(* Logix 5000 project; controller TCP vendor 1 type 14 code 178 rev 35.12; software revision 35.01 *)

TASK MainTask (continuous, watchdog 500 ms) : MainProgram, TCP_Connection
TASK SafetyTask (periodic, rate 20 ms, priority 10, watchdog 20 ms, safety) : SafetyProgram

MODULES
   Local : vendor 1 type 14 code 178 (Compact 0, rev 35.12)
END_MODULES

TYPE MSG_CreateParameters :
STRUCT
   Type : DINT;   // 1 - TCP ; 2 - UPD
   Addr : MSG_SockAddr;   // Address for the Socket
END_STRUCT
END_TYPE

TYPE MSG_OpenConnectionParameters :
STRUCT
   TimeOut : DINT;   // Timeout in milliseconds
   DestAddr : STRING;   // Hostname or IP adress (ex : 10.88.81.10?port=2813 OR name?port=2813)
END_STRUCT
END_TYPE

TYPE MSG_ReadParameters :
STRUCT
   TimeOut : DINT;   // TimeOut in milliseconds
   BufLen : DINT;   // Number of bytes of data to receive
END_STRUCT
END_TYPE

TYPE MSG_ReadResponse :
STRUCT
   FromAddr : MSG_SockAddr;   // A user-defined structure that can contain the address of the device that sends UDP data. This structure is populated from the end device. For TCP or UDP with OpenConnection, this structure is not used and contains all zeros. The TCP connection conveys all remote address information
   BufLen : DINT;   // Contains the number of bytes of data received
   Buf : SINT[484];   // Contains the data. This number must be large enough to contain the maximum amount of data expected. For a standard connection, the maximum is SINT[484]. For a large connection, the maximum is SINT [3984].
END_STRUCT
END_TYPE

TYPE MSG_SockAddr :
STRUCT
   Family : INT;   // Adress Family Must be 2
   Port : INT;   // Port Number - If random needed use 0
   Addr : DINT;   // IP Address - Each Byte are separated for xxx.xxx.xxx.xxx
END_STRUCT
END_TYPE

TYPE MSG_WriteParameters :
STRUCT
   TimeOut : DINT;   // TimeOut in milliseconds
   ToAddr : MSG_SockAddr;   // Structure that contains the address to which to write UDP data. For TCP or UDP with OpenConnection, this structure is not used and contains all zeros. The TCP connection conveys all required remote address information.
   BufLen : DINT;   // Specify the number of bytes of data to write
   Buf : SINT[472];   // Contains the data. This number must be large enough to contain the maximum amount of data expected. For a standard connection, the maximum is SINT[472]. For a large connection, the maximum is SINT [3972].
END_STRUCT
END_TYPE

VAR_GLOBAL   (* controller tags *)
   Destination_Element_Read_Request : MSG_ReadResponse := (FromAddr.Family := 2, Buf[0] := 78, Buf[1] := 75, Buf[2] := 80, Buf[3] := 49, Buf[9] := 1, Buf[12] := 107, Buf[13] := 99, Buf[14] := 111, Buf[21] := 3, Buf[25] := 1, Buf[29] := 1, Buf[34] := 15, Buf[35] := -125, Buf[36] := -20, Buf[37] := -78, Buf[38] := 50, Buf[39] := 54, Buf[40] := 48, Buf[41] := 51, Buf[42] := 48, Buf[43] := 52, Buf[44] := 48, Buf[45] := 53, Buf[46] := 48, Buf[61] := 3, Buf[63] := -115, Buf[64] := 23, Buf[65] := 112, Buf[66] := 19, Buf[67] := -119, Buf[75] := 48, Buf[76] := 7, Buf[77] := -47, Buf[79] := 60, Buf[80] := 107, Buf[81] := 99, Buf[82] := 111, Buf[89] := 3, Buf[91] := 1, Buf[92] := -20, Buf[93] := -95, Buf[94] := 50, Buf[95] := 54, Buf[96] := 48, Buf[97] := 51, Buf[98] := 48, Buf[99] := 52, Buf[100] := 48, Buf[101] := 51, Buf[102] := 51, Buf[117] := 93, Buf[119] := -115, Buf[120] := 2, Buf[121] := 89, Buf[122] := 19, Buf[123] := -119, Buf[126] := 4, Buf[127] := -52, Buf[130] := 5,
        Buf[131] := 8, Buf[132] := 7, Buf[133] := -41, Buf[135] := 60, Buf[136] := 107, Buf[137] := 99, Buf[138] := 111, Buf[145] := 3, Buf[147] := 2, Buf[148] := 107, Buf[149] := 99, Buf[150] := 111, Buf[157] := 3, Buf[159] := 2, Buf[160] := -20, Buf[161] := -95, Buf[162] := 50, Buf[163] := 54, Buf[164] := 48, Buf[165] := 51, Buf[166] := 48, Buf[167] := 52, Buf[168] := 48, Buf[169] := 51, Buf[170] := 51, Buf[185] := 93, Buf[187] := -115, Buf[188] := 2, Buf[189] := 89, Buf[190] := 19, Buf[191] := -119, Buf[194] := 5, Buf[195] := 59, Buf[198] := 5, Buf[199] := 119, Buf[200] := 7, Buf[201] := -41, Buf[203] := 60, Buf[204] := 107, Buf[205] := 99, Buf[206] := 111, Buf[213] := 3, Buf[215] := 3, Buf[216] := 107, Buf[217] := 99, Buf[218] := 111, Buf[225] := 3, Buf[227] := 3, Buf[229] := 4, Buf[233] := 4, Buf[238] := 15, Buf[239] := -125, Buf[240] := -20, Buf[241] := -95, Buf[242] := 50, Buf[243] := 54, Buf[244] := 48, Buf[245] := 51, Buf[246] := 48, Buf[247] := 52,
        Buf[248] := 48, Buf[249] := 51, Buf[250] := 51, Buf[265] := 93, Buf[267] := -115, Buf[268] := 2, Buf[269] := 89, Buf[270] := 19, Buf[271] := -119, Buf[274] := 9, Buf[275] := -13, Buf[278] := 10, Buf[279] := 47, Buf[280] := 7, Buf[281] := -41, Buf[283] := 60, Buf[284] := 107, Buf[285] := 99, Buf[286] := 111, Buf[293] := 3, Buf[295] := 4, Buf[297] := 5, Buf[301] := 5, Buf[306] := 15, Buf[307] := -125, Buf[308] := -20, Buf[309] := -95, Buf[310] := 50, Buf[311] := 54, Buf[312] := 48, Buf[313] := 51, Buf[314] := 48, Buf[315] := 52, Buf[316] := 48, Buf[317] := 51, Buf[318] := 51, Buf[333] := 93, Buf[335] := -115, Buf[336] := 2, Buf[337] := 89, Buf[338] := 19, Buf[339] := -119, Buf[342] := 13, Buf[343] := -50, Buf[346] := 14, Buf[347] := 10, Buf[348] := 7, Buf[349] := -41, Buf[351] := 60, Buf[352] := 107, Buf[353] := 99, Buf[354] := 111, Buf[361] := 3, Buf[363] := 5, Buf[365] := 6, Buf[369] := 6, Buf[374] := 15, Buf[375] := -125, Buf[376] := -20, Buf[377] := -95,
        Buf[378] := 50, Buf[379] := 54, Buf[380] := 48, Buf[381] := 51, Buf[382] := 48, Buf[383] := 52, Buf[384] := 48, Buf[385] := 51, Buf[386] := 51, Buf[401] := 93, Buf[403] := -115, Buf[404] := 2, Buf[405] := 89, Buf[406] := 19, Buf[407] := -119, Buf[410] := 14, Buf[411] := 25, Buf[414] := 14, Buf[415] := 85, Buf[416] := 7, Buf[417] := -41, Buf[419] := 60, Buf[420] := 107, Buf[421] := 99, Buf[422] := 111, Buf[429] := 3, Buf[431] := 6, Buf[433] := 7, Buf[437] := 7, Buf[442] := 15, Buf[443] := -125, Buf[444] := -20, Buf[445] := -95, Buf[446] := 50, Buf[447] := 54, Buf[448] := 48, Buf[449] := 51, Buf[450] := 48, Buf[451] := 52, Buf[452] := 48, Buf[453] := 51, Buf[454] := 51, Buf[469] := 93, Buf[471] := -115, Buf[472] := 2, Buf[473] := 89, Buf[474] := 19, Buf[475] := -119, Buf[478] := 15, Buf[479] := -31, Buf[482] := 16, Buf[483] := 29);
   Destination_Element_Write_Request : DINT := 48;   // Lenght of the Data written
   Destination_Element_Write_Request_Payloa : DINT := 48;   // Lenght of the Data written
   Instance_OPTP : DINT := 21276;
   MSG_Create_Socket : MESSAGE;
        MessageParameters(ServiceCode := 16#004b, LocalElement := Source_Element_Create_Socket, DestinationTag := Instance_OPTP, ...)
   MSG_Delete_All_Socket : MESSAGE;
        MessageParameters(ServiceCode := 16#0051, ...)
   MSG_Open_Connection : MESSAGE;
        MessageParameters(ServiceCode := 16#004c, LocalElement := Source_Element_Open_Connection, ...)
   MSG_Read_Request : MESSAGE;
        MessageParameters(ServiceCode := 16#004d, LocalElement := Source_Element_Read_Request, DestinationTag := Destination_Element_Read_Request, ...)
   MSG_Write_Request : MESSAGE;
        MessageParameters(ServiceCode := 16#004e, LocalElement := Source_Element_Write_Request, DestinationTag := Destination_Element_Write_Request, ...)
   MSG_Write_Request_Payload : MESSAGE;
        MessageParameters(ServiceCode := 16#004e, LocalElement := Source_Element_Write_Request_Payload, DestinationTag := Destination_Element_Write_Request_Payloa, ...)
   Source_Element_Create_Socket : MSG_CreateParameters := (Type := 1, Addr.Family := 2);   // Source parameters for MSG Create Socket
   Source_Element_Open_Connection : MSG_OpenConnectionParameters := (TimeOut := 5000, DestAddr := '192.120.0.203?port=5010$00');
   Source_Element_Read_Request : MSG_ReadParameters := (TimeOut := 3000, BufLen := 484);
   Source_Element_Write_Request : MSG_WriteParameters := (TimeOut := 5000, BufLen := 8, Buf[0] := 78, Buf[1] := 75, Buf[2] := 80, Buf[3] := 49, Buf[4] := 57, Buf[5] := 57, Buf[6] := 57, Buf[7] := 57);
   Source_Element_Write_Request_Payload : MSG_WriteParameters := (TimeOut := 5000, BufLen := 7, Buf[0] := 98, Buf[1] := 105, Buf[2] := 103, Buf[3] := 78, Buf[4] := 75, Buf[5] := 80, Buf[6] := 50);
END_VAR

PROGRAM MainProgram   (* main routine MainRoutine *)

ROUTINE MainRoutine   (* ladder *)
END_ROUTINE
END_PROGRAM

PROGRAM SafetyProgram   (* main routine MainRoutine, safety *)

ROUTINE MainRoutine   (* ladder *)
END_ROUTINE
END_PROGRAM

PROGRAM TCP_Connection   (* main routine Main *)
VAR
   Action_000 : SFC_ACTION := (Status := 16#0020_0000, PauseTimer := 1);
   Action_001 : SFC_ACTION := (Status := 16#0020_0000, PauseTimer := 1);
   Action_002 : SFC_ACTION := (Status := 16#0020_0000, PauseTimer := 1);
   Action_003 : SFC_ACTION := (Status := 16#0020_0000, PauseTimer := 1);
   Action_004 : SFC_ACTION := (Status := 16#0020_0000, PauseTimer := 1);
   Action_005 : SFC_ACTION := (Status := 16#0020_0000, PauseTimer := 1);
   Action_006 : SFC_ACTION := (Status := 16#0020_0000, PauseTimer := 1);
   Action_007 : SFC_ACTION := (Status := 16#0020_0000, PauseTimer := 1);
   Action_008 : SFC_ACTION := (Status := 16#0020_0000, PauseTimer := 1);
   Convert_ok : BOOL;
   FALSE : BOOL; {constant}
   Footer_Invalid : BOOL;
   Footer_Valid : BOOL;   // M
   Header_At_Zero : BOOL;   // M
   Header_Found : BOOL;   // M
   Header_Pos : DINT;   // M B
   Header_Ready : BOOL;   // M
   Header_Send : BOOL;   // M
   Header_Valid : BOOL;   // M
   I_Size_Payload : DINT;   // M B
   ind : DINT;
   Init_Done : BOOL;   // M
   Invalide_Size_Format : BOOL;   // M
   NEKO : BOOL;   // B
   No_Header : BOOL;
   ONS : BOOL[32];
        [0]   // used
        [1]   // used
        [2]   // used
   Open_Connection : BOOL;   // M
   Open_started : BOOL := 1;   // M
   Payload_buffer : SINT[4096];   // M B
   Read_Done : BOOL;   // M
   Request_to_send : BOOL;   // M B
   Reset_Error : BOOL;   // M B
   Rx_Buffer : SINT[4096];   // M B
   Rx_Count : DINT;   // M B
   Rx_Update : BOOL;
   S00_Init : SFC_STEP := (Status := 16#0020_0000, PauseTimer := 1);
   S100_CHECK_FOOTER : SFC_STEP := (Status := 16#0020_0000, PauseTimer := 1);
   S10_IDLE : SFC_STEP := (Status := 16#0020_0000, PauseTimer := 1);
   S110_EXTRACT : SFC_STEP := (Status := 16#0020_0000, PauseTimer := 1);
   S120_PROCESS : SFC_STEP := (Status := 16#0020_0000, PauseTimer := 1);
   S130_RESYNC : SFC_STEP := (Status := 16#0020_0000, PauseTimer := 1);
   S20_Write : SFC_STEP := (Status := 16#0020_0000, PauseTimer := 1);
   S30_WAIT_DATA : SFC_STEP := (Status := 16#0020_0000, PauseTimer := 1);
   S40_APPEND_DATA : SFC_STEP := (Status := 16#0020_0000, PauseTimer := 1);
   S50_FIIND_HEADER : SFC_STEP := (Status := 16#0020_0000, PauseTimer := 1);
   S60_CLEAN_BUFFER : SFC_STEP := (Status := 16#0020_0000, PauseTimer := 1);
   S70_WAIT_HEADER : SFC_STEP := (Status := 16#0020_0000, PauseTimer := 1);
   S80_CHECK_HEADER : SFC_STEP := (Status := 16#0020_0000, PauseTimer := 1);
   S900_ERROR : SFC_STEP := (Status := 16#0020_0000, PauseTimer := 1);
   S90_WAIT_FRAME : SFC_STEP := (Status := 16#0020_0000, PauseTimer := 1);
   Signature_False : BOOL;   // M
   Size_Overflow : BOOL;   // M
   Size_Payload : STRING;   // M B
   Socket_Create : BOOL;   // M
   T00A10 : BOOL;
   T00A900 : BOOL;
   T100A110 : BOOL;
   T100A130 : BOOL;
   T10A20 : BOOL;
   T110A120 : BOOL;
   T120A10 : BOOL;
   T120A50 : BOOL;
   T130A30 : BOOL;
   T130A50 : BOOL;
   T20A30 : BOOL;
   T20A900 : BOOL;
   T30A40 : BOOL;
   T30A401 : BOOL;
   T30A900 : BOOL;
   T40A50 : BOOL;
   T50A30 : BOOL;
   T50A60 : BOOL;
   T50A70 : BOOL;
   T60A80 : BOOL;
   T70A30 : BOOL;
   T70A80 : BOOL;
   T80A130 : BOOL;
   T80A90 : BOOL;
   T900A00 : BOOL;
   T90A100 : BOOL;
   T90A30 : BOOL;
   TRUE : BOOL := 1; {constant}
   Write_Done : BOOL;   // M
END_VAR

ROUTINE Graphe_Etat   (* sequential function chart *)
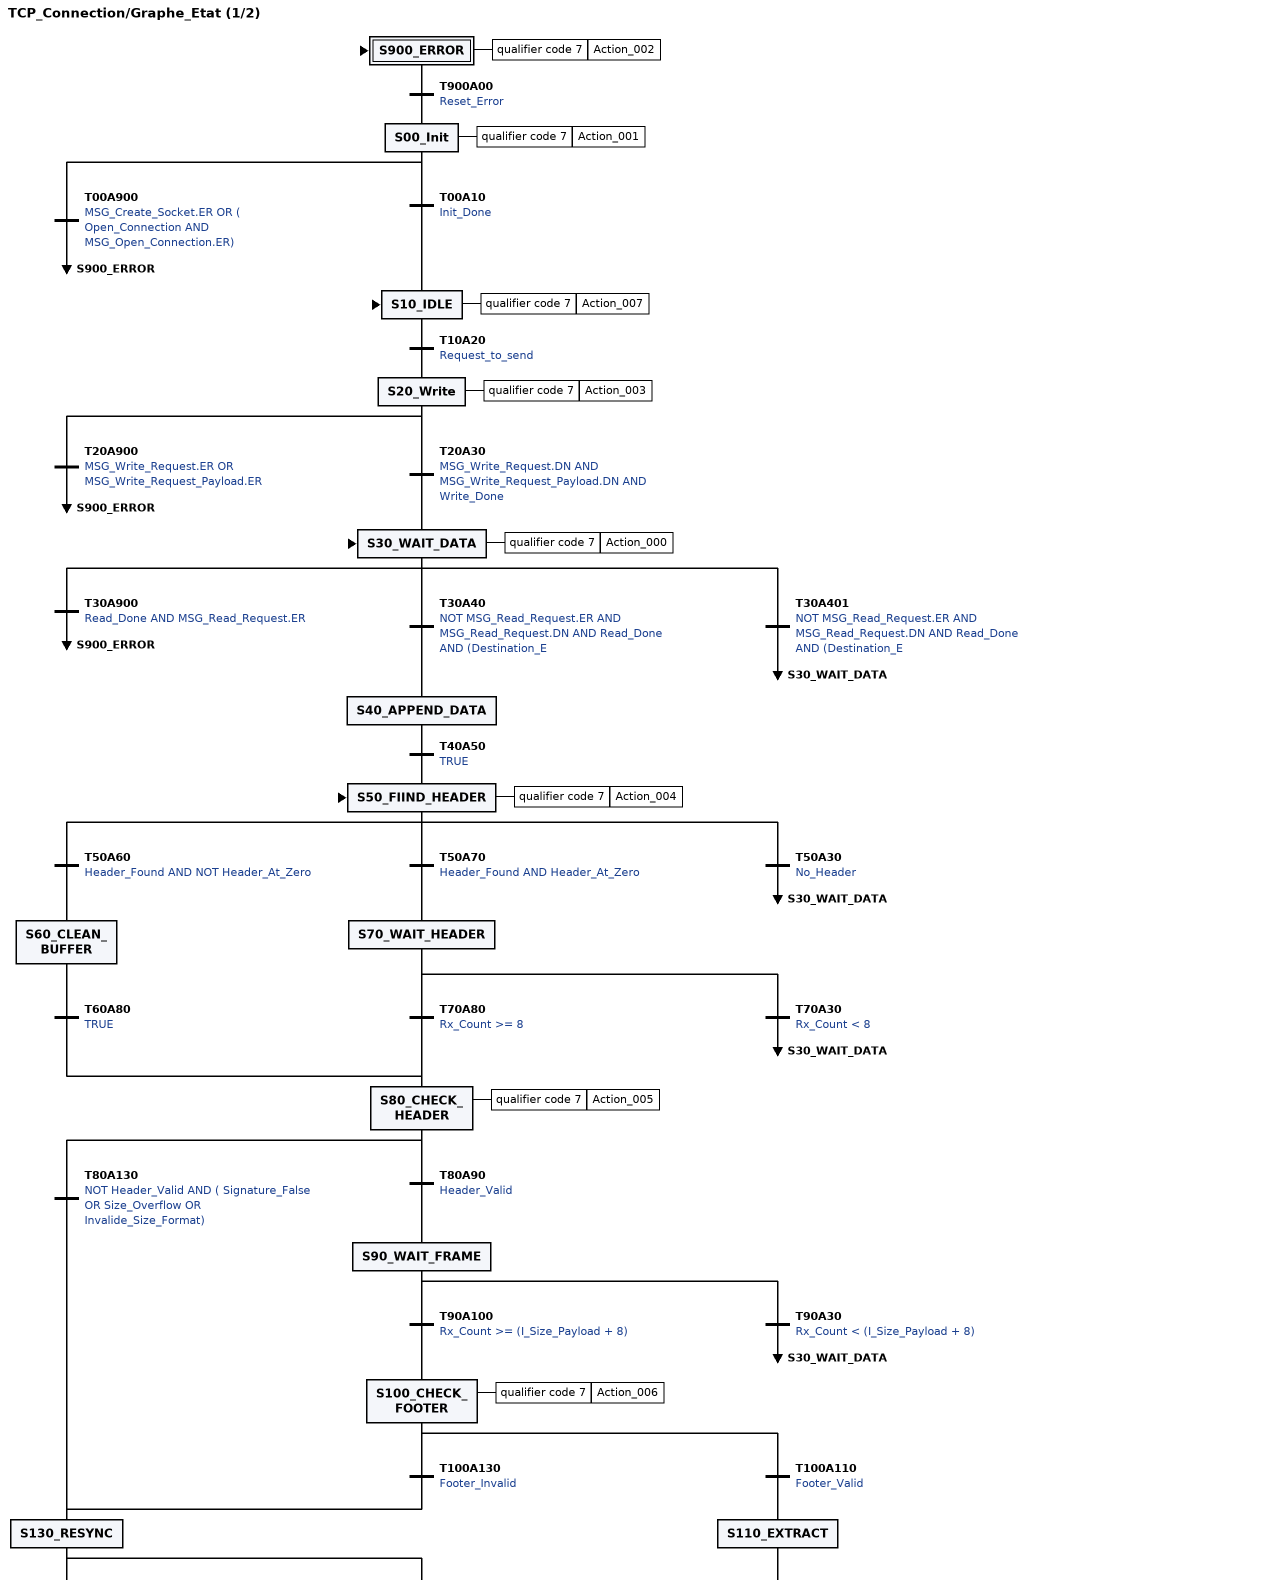
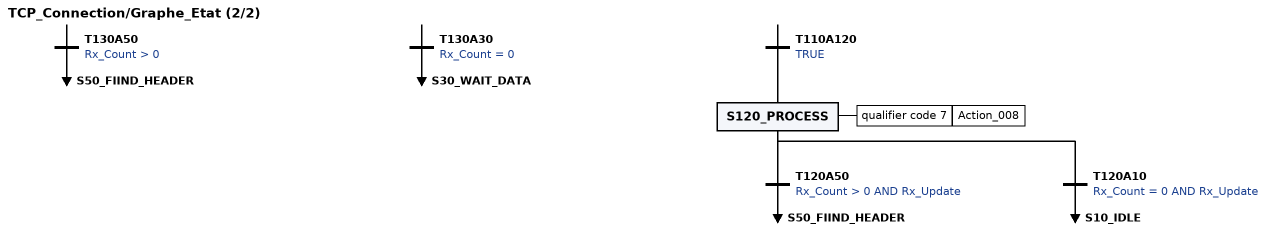
   // RESET ALL
   INITIAL_STEP S900_ERROR:
      ACTION Action_002 (qualifier code 7):
         Reset_Error := 0;
      END_ACTION
   END_STEP
   TRANSITION T900A00 FROM S900_ERROR TO S00_Init
      := Reset_Error
   END_TRANSITION
   STEP S00_Init:
      ACTION Action_001 (qualifier code 7):
         Socket_Create := 0;
         Open_started := 0;
         Open_Connection := 0;
         Init_Done := 0;
      END_ACTION
   END_STEP
   TRANSITION T00A900 FROM S00_Init TO S900_ERROR
      := MSG_Create_Socket.ER OR (
         Open_Connection AND
         MSG_Open_Connection.ER)
   END_TRANSITION
   TRANSITION T00A10 FROM S00_Init TO S10_IDLE
      := Init_Done
   END_TRANSITION
   STEP S10_IDLE:
      ACTION Action_007 (qualifier code 7):
         Rx_Count := 0;
         Request_to_send := 0;
      END_ACTION
   END_STEP
   TRANSITION T10A20 FROM S10_IDLE TO S20_Write
      := Request_to_send
   END_TRANSITION
   STEP S20_Write:
      ACTION Action_003 (qualifier code 7):
         Convert_ok := 0;
         Header_Send := 0;
         Write_Done := 0;
      END_ACTION
   END_STEP
   TRANSITION T20A900 FROM S20_Write TO S900_ERROR
      := MSG_Write_Request.ER OR
         MSG_Write_Request_Payload.ER
   END_TRANSITION
   TRANSITION T20A30 FROM S20_Write TO S30_WAIT_DATA
      := MSG_Write_Request.DN AND
         MSG_Write_Request_Payload.DN AND
         Write_Done
         
   END_TRANSITION
   STEP S30_WAIT_DATA:
      ACTION Action_000 (qualifier code 7):
         Read_Done := 0;
         Destination_Element_Read_Request.BufLen :=0;
      END_ACTION
   END_STEP
   TRANSITION T30A40 FROM S30_WAIT_DATA TO S40_APPEND_DATA
      := NOT MSG_Read_Request.ER AND
         MSG_Read_Request.DN AND
         Read_Done AND
         (Destination_Element_Read_Request.BufLen > 0)
   END_TRANSITION
   TRANSITION T30A401 FROM S30_WAIT_DATA TO S30_WAIT_DATA
      := NOT MSG_Read_Request.ER AND
         MSG_Read_Request.DN AND
         Read_Done AND
         (Destination_Element_Read_Request.BufLen = 0)
   END_TRANSITION
   TRANSITION T30A900 FROM S30_WAIT_DATA TO S900_ERROR
      := Read_Done AND
         MSG_Read_Request.ER
   END_TRANSITION
   STEP S40_APPEND_DATA:
   END_STEP
   TRANSITION T40A50 FROM S40_APPEND_DATA TO S50_FIIND_HEADER
      := TRUE
         
   END_TRANSITION
   STEP S50_FIIND_HEADER:
      ACTION Action_004 (qualifier code 7):
         Header_Found := 0;
         Header_At_Zero := 0;
         Header_Pos := 0;
         No_Header := 0;
      END_ACTION
   END_STEP
   TRANSITION T50A60 FROM S50_FIIND_HEADER TO S60_CLEAN_BUFFER
      := Header_Found AND NOT
         Header_At_Zero
   END_TRANSITION
   TRANSITION T50A70 FROM S50_FIIND_HEADER TO S70_WAIT_HEADER
      := Header_Found AND
         Header_At_Zero
         
         
   END_TRANSITION
   TRANSITION T50A30 FROM S50_FIIND_HEADER TO S30_WAIT_DATA
      := No_Header
   END_TRANSITION
   STEP S60_CLEAN_BUFFER:
   END_STEP
   STEP S70_WAIT_HEADER:
   END_STEP
   TRANSITION T60A80 FROM S60_CLEAN_BUFFER TO S80_CHECK_HEADER
      := TRUE
   END_TRANSITION
   TRANSITION T70A80 FROM S70_WAIT_HEADER TO S80_CHECK_HEADER
      := Rx_Count >= 8
   END_TRANSITION
   TRANSITION T70A30 FROM S70_WAIT_HEADER TO S30_WAIT_DATA
      := Rx_Count < 8
   END_TRANSITION
   STEP S80_CHECK_HEADER:
      ACTION Action_005 (qualifier code 7):
         Invalide_Size_Format := 0;
         Size_Overflow := 0;
         Header_Valid := 0;
         Signature_False := 0;
      END_ACTION
   END_STEP
   TRANSITION T80A130 FROM S80_CHECK_HEADER TO S130_RESYNC
      := NOT Header_Valid AND (
         Signature_False OR
         Size_Overflow OR
         Invalide_Size_Format)
   END_TRANSITION
   TRANSITION T80A90 FROM S80_CHECK_HEADER TO S90_WAIT_FRAME
      := Header_Valid
   END_TRANSITION
   STEP S90_WAIT_FRAME:
   END_STEP
   TRANSITION T90A30 FROM S90_WAIT_FRAME TO S30_WAIT_DATA
      := Rx_Count < (I_Size_Payload + 8)
   END_TRANSITION
   TRANSITION T90A100 FROM S90_WAIT_FRAME TO S100_CHECK_FOOTER
      := Rx_Count >= (I_Size_Payload + 8)
   END_TRANSITION
   STEP S100_CHECK_FOOTER:
      ACTION Action_006 (qualifier code 7):
         Footer_Valid := 0;
         Footer_Invalid := 0;
      END_ACTION
   END_STEP
   TRANSITION T100A130 FROM S100_CHECK_FOOTER TO S130_RESYNC
      := Footer_Invalid
   END_TRANSITION
   TRANSITION T100A110 FROM S100_CHECK_FOOTER TO S110_EXTRACT
      := Footer_Valid
   END_TRANSITION
   STEP S130_RESYNC:
   END_STEP
   STEP S110_EXTRACT:
   END_STEP
   TRANSITION T130A50 FROM S130_RESYNC TO S50_FIIND_HEADER
      := Rx_Count > 0
   END_TRANSITION
   TRANSITION T130A30 FROM S130_RESYNC TO S30_WAIT_DATA
      := Rx_Count = 0
   END_TRANSITION
   TRANSITION T110A120 FROM S110_EXTRACT TO S120_PROCESS
      := TRUE
   END_TRANSITION
   STEP S120_PROCESS:
      ACTION Action_008 (qualifier code 7):
         Rx_Update := 0;
      END_ACTION
   END_STEP
   TRANSITION T120A50 FROM S120_PROCESS TO S50_FIIND_HEADER
      := Rx_Count > 0 AND
         Rx_Update
   END_TRANSITION
   TRANSITION T120A10 FROM S120_PROCESS TO S10_IDLE
      := Rx_Count = 0 AND
         Rx_Update
         
   END_TRANSITION
END_ROUTINE

ROUTINE Main   (* ladder *)
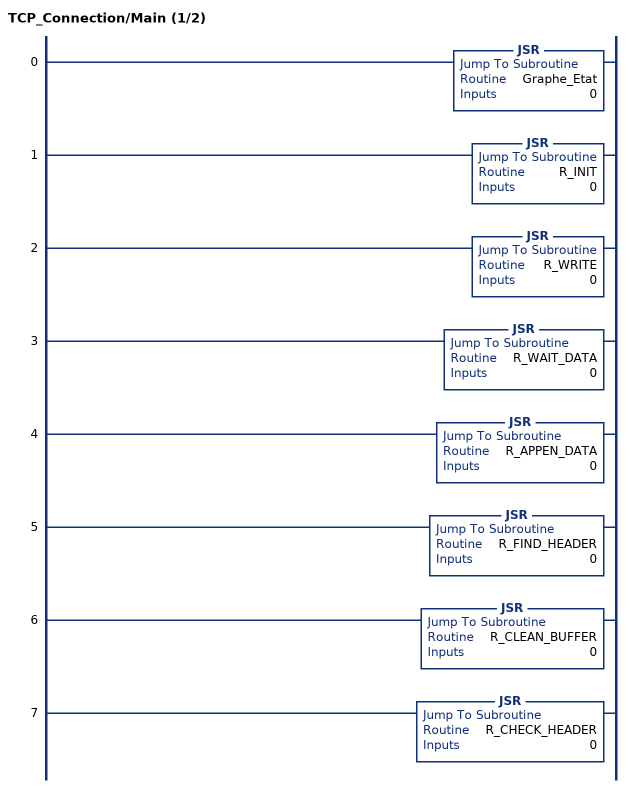
   0: JSR(Graphe_Etat,0);
   1: JSR(R_INIT,0);
   2: JSR(R_WRITE,0);
   3: JSR(R_WAIT_DATA,0);
   4: JSR(R_APPEN_DATA,0);
   5: JSR(R_FIND_HEADER,0);
   6: JSR(R_CLEAN_BUFFER,0);
   7: JSR(R_CHECK_HEADER,0);
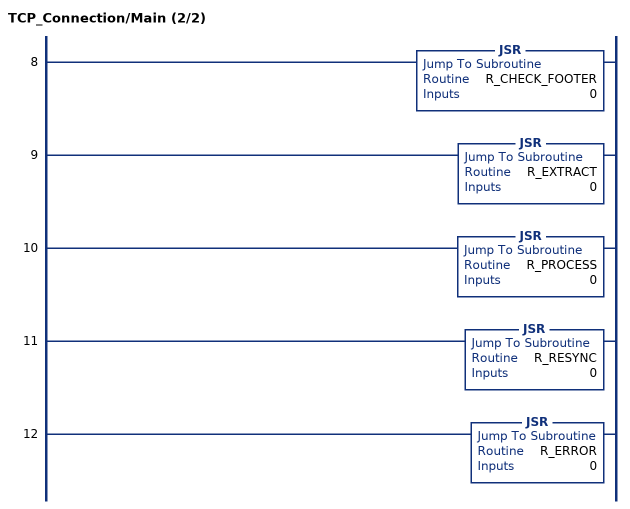
   8: JSR(R_CHECK_FOOTER,0);
   9: JSR(R_EXTRACT,0);
   10: JSR(R_PROCESS,0);
   11: JSR(R_RESYNC,0);
   12: JSR(R_ERROR,0);
END_ROUTINE

ROUTINE R_APPEN_DATA   (* structured text *)
   IF S40_APPEND_DATA.SA THEN
   	for ind := 0 to (Destination_Element_Read_Request.BufLen - 1) do
   		Rx_Buffer[Rx_Count + ind] := Destination_Element_Read_Request.Buf[ind];
   	end_for;
   	Rx_Count := Rx_Count + Destination_Element_Read_Request.BufLen;
   ELSE
   END_IF;
END_ROUTINE

ROUTINE R_CHECK_FOOTER   (* structured text *)
   IF S100_CHECK_FOOTER.SA THEN
   	IF Rx_Buffer[Rx_Count - 4] = 78 AND Rx_Buffer[Rx_Count - 3] = 75 AND
   	   Rx_Buffer[Rx_Count - 2] = 80 AND Rx_Buffer[Rx_Count - 1] = 50 THEN
   	   Footer_Valid := 1;
   	   Footer_Invalid := 0;
   
   	ELSE
   		Footer_Invalid := 1;
   		Footer_Valid := 0;
   	END_IF;
   ELSE
   
   END_IF;
   
END_ROUTINE

ROUTINE R_CHECK_HEADER   (* structured text *)
   IF S80_CHECK_HEADER.SA THEN
   	IF Rx_Buffer[0] = 78 AND Rx_Buffer[1] = 75 AND Rx_Buffer[2] = 80 AND Rx_Buffer[3] = 49 THEN
   		FOR ind := 4 TO 7 DO
   			Size_Payload.DATA[ind - 4] := Rx_Buffer[ind];
   		END_FOR;
   		Size_Payload.LEN := 4;
   
   		// Copy into a STRING buffer for convertion purpuse
   		FOR ind := 0 TO 3 DO
   			//Check that the ASCII format refer to a number
   			IF Size_Payload.DATA[ind] > 57 OR Size_Payload.DATA[ind] < 48 THEN
   				Invalide_Size_Format := 1;
   				EXIT;
   			ELSE
   				Invalide_Size_Format := 0;
   			END_IF;
   		END_FOR;
   		IF NOT Invalide_Size_Format THEN
   			//Convert to a DINT then we check that the size is not bigger than our Rx_Buffer
   			STOD(Size_Payload, I_Size_Payload);
   			IF I_Size_Payload > 4096 THEN
   				Size_Overflow := 1;
   				Header_Valid := 0;
   			ELSE
   				Size_Overflow := 0;
   				Header_Valid := 1;
   			END_IF;
   		ELSE
   			// Nothing to do because invalide format
   		END_IF;
   	ELSE
   		Signature_False := 1;
   	END_IF;
   ELSE
   
   END_IF;
END_ROUTINE

ROUTINE R_CLEAN_BUFFER   (* structured text *)
   IF S60_CLEAN_BUFFER.FS THEN
   	FOR ind := 0 TO (Rx_Count - 1 - Header_Pos) DO
   		Rx_Buffer[ind] := Rx_Buffer[Header_Pos + ind];
   	END_FOR;
   	Rx_Count := Rx_Count - Header_Pos;
   ELSE
   
   END_IF;
END_ROUTINE

ROUTINE R_ERROR   (* ladder *)
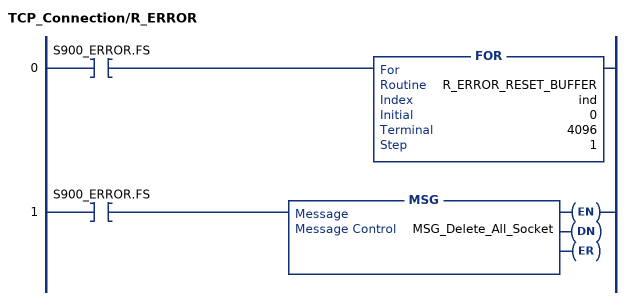
   0: XIC(S900_ERROR.FS)FOR(R_ERROR_RESET_BUFFER,ind,0,4096,1);
   1: XIC(S900_ERROR.FS)MSG(MSG_Delete_All_Socket);
END_ROUTINE

ROUTINE R_ERROR_RESET_BUFFER   (* ladder *)
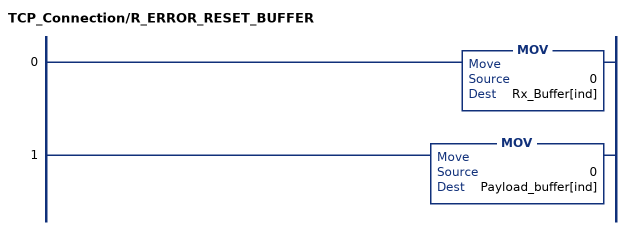
   0: MOV(0,Rx_Buffer[ind]);
   1: MOV(0,Payload_buffer[ind]);
END_ROUTINE

ROUTINE R_EXTRACT   (* structured text *)
   IF S110_EXTRACT.SA THEN
   	FOR ind := 0 TO (Rx_Count - 8 - 4 - 1) DO  //8 for header 4 for footer
   		Payload_buffer[ind] := Rx_Buffer[8 + ind];
   	END_FOR;
   ELSE
   
   END_IF;
END_ROUTINE

ROUTINE R_FIND_HEADER   (* structured text *)
   IF S50_FIIND_HEADER.SA THEN
   	FOR ind := 0 TO (Rx_Count - 4) DO
   		IF Rx_Buffer[ind] = 78 AND Rx_Buffer[ind + 1] = 75 AND Rx_Buffer[ind + 2] = 80 AND Rx_Buffer[ind + 3] = 49 THEN
   			Header_Found := 1;
   			No_Header := 0;
   			Header_Pos := ind;
   			IF Header_Pos = 0 THEN
   				Header_At_Zero := 1;
   			END_IF;
   			EXIT;
   		ELSE
   
   		END_IF;
   	END_FOR;
   	IF ind >= (Rx_Count - 4) then
   		Header_Found := 0;
   		No_Header := 1;
   	END_IF;
   ELSE
   
   END_IF;
END_ROUTINE

ROUTINE R_INIT   (* ladder *)
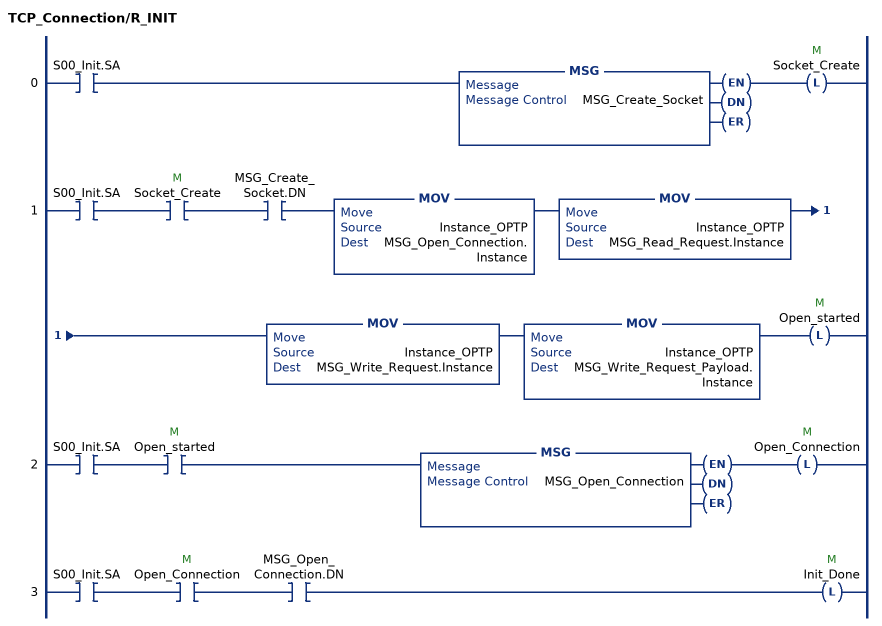
   0: XIC(S00_Init.SA)MSG(MSG_Create_Socket)OTL(Socket_Create);
   1: XIC(S00_Init.SA)XIC(Socket_Create)XIC(MSG_Create_Socket.DN)MOV(Instance_OPTP,MSG_Open_Connection.Instance)MOV(Instance_OPTP,MSG_Read_Request.Instance)MOV(Instance_OPTP,MSG_Write_Request.Instance)MOV(Instance_OPTP,MSG_Write_Request_Payload.Instance)OTL(Open_started);
   2: XIC(S00_Init.SA)XIC(Open_started)MSG(MSG_Open_Connection)OTL(Open_Connection);
   3: XIC(S00_Init.SA)XIC(Open_Connection)XIC(MSG_Open_Connection.DN)OTL(Init_Done);
END_ROUTINE

ROUTINE R_PROCESS   (* structured text *)
   //No DATA to process now
   IF S120_PROCESS.SA AND NOT Rx_Update THEN
   	Rx_Count := Rx_Count - 8 - I_Size_Payload;
   	Rx_Update := 1;
   ELSE
   END_iF;
END_ROUTINE

ROUTINE R_RESYNC   (* structured text *)
   IF S130_RESYNC.FS THEN
   
   ELSE
   
   END_IF;
END_ROUTINE

ROUTINE R_WAIT_DATA   (* ladder *)
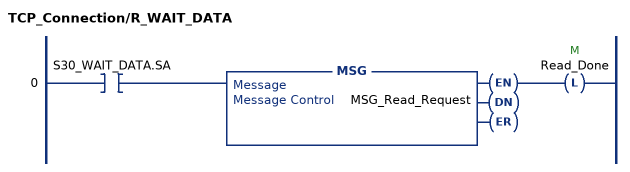
   0: XIC(S30_WAIT_DATA.SA)MSG(MSG_Read_Request)OTL(Read_Done);
END_ROUTINE

ROUTINE R_WRITE   (* ladder *)
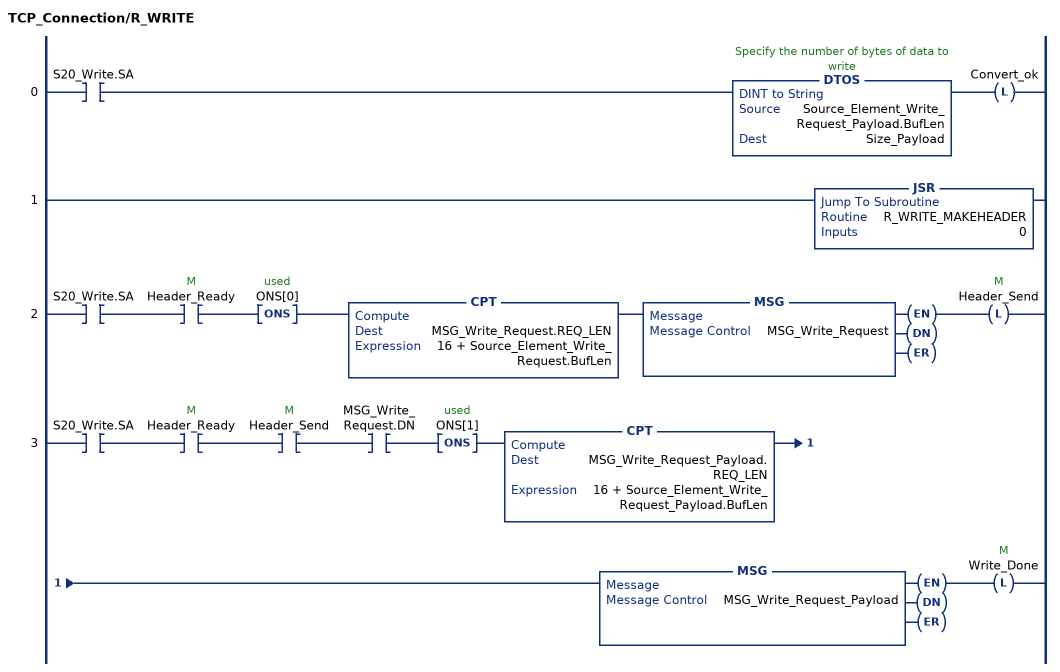
   0: XIC(S20_Write.SA)DTOS(Source_Element_Write_Request_Payload.BufLen,Size_Payload)OTL(Convert_ok);
   1: JSR(R_WRITE_MAKEHEADER,0);
   2: XIC(S20_Write.SA)XIC(Header_Ready)ONS(ONS[0])CPT(MSG_Write_Request.REQ_LEN,16 + Source_Element_Write_Request.BufLen)MSG(MSG_Write_Request)OTL(Header_Send);
   3: XIC(S20_Write.SA)XIC(Header_Ready)XIC(Header_Send)XIC(MSG_Write_Request.DN)ONS(ONS[1])CPT(MSG_Write_Request_Payload.REQ_LEN,16 + Source_Element_Write_Request_Payload.BufLen)MSG(MSG_Write_Request_Payload)OTL(Write_Done);
END_ROUTINE

ROUTINE R_WRITE_MAKEHEADER   (* structured text *)
   IF S20_Write.SA AND Convert_ok THEN
   
   	FOR ind := 1 TO Size_Payload.LEN DO
   	    Source_Element_Write_Request.Buf[4 + (4 - Size_Payload.LEN) + (ind - 1)] := Size_Payload.DATA[ind - 1];
   	END_FOR;
   
   	FOR ind := 1 TO (4 - Size_Payload.LEN) DO
   	    Source_Element_Write_Request.Buf[4 + (ind - 1)] := 48;
   	END_FOR;
   
   	Header_Ready := 1;
   ELSE
   
   END_IF;
END_ROUTINE
END_PROGRAM
